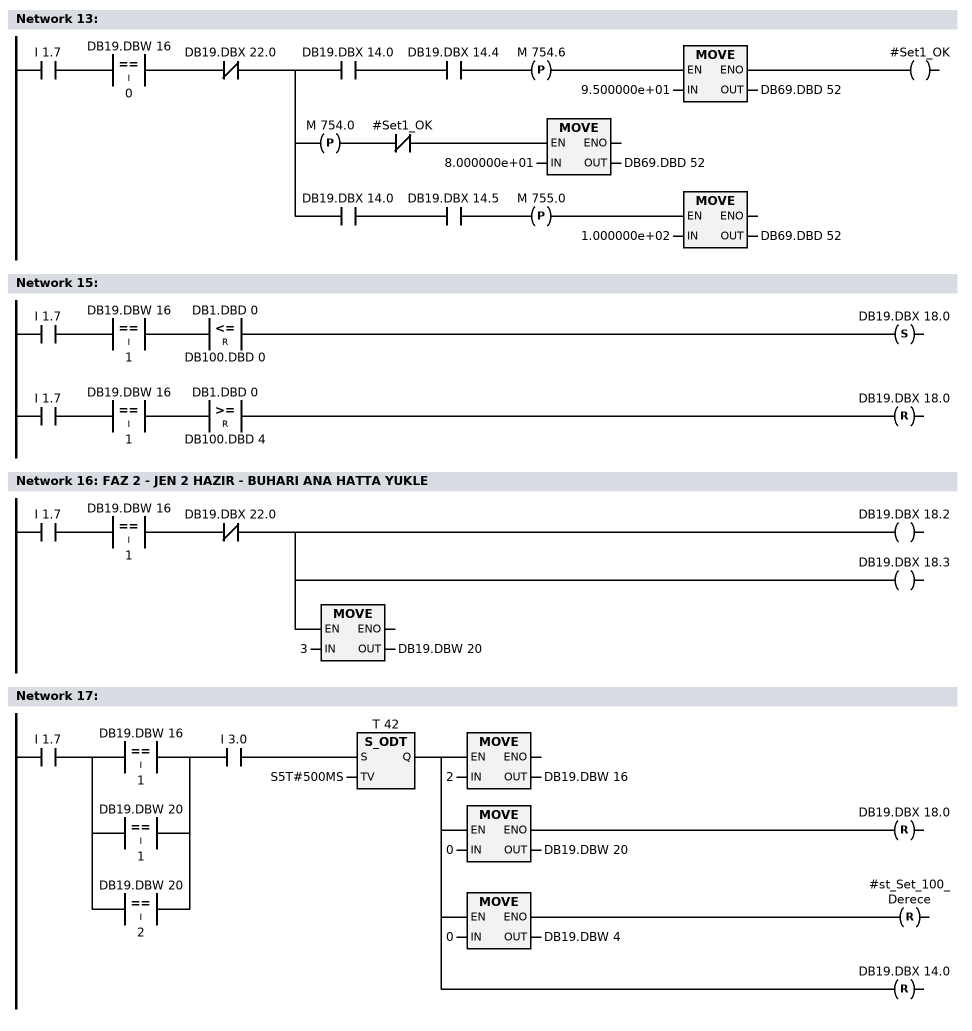
NETWORK
TITLE =
//-Sicaklik set 1 e geldiginde vana kapanma orani 5'e kadar düsüyor
//-Sicaklik set 2 e geldiginde vana kapanma orani 0'a kadar dusecek
//
//m754.0
//
      A     I 1.7;
      A(;
      L     DB19.DBW 16;
      L     0;
      ==I;
      );
      AN    DB19.DBX 22.0;
      =     L 2.0;
      A     L 2.0;
      A     DB19.DBX 14.0;
      A     DB19.DBX 14.4;
      FP    M 754.6;
      JNB   _00b;
      L     9.500000e+01;
      T     DB69.DBD 52;
      SET;
      SAVE;
      CLR;
_00b: A     BR;
      =     #Set1_OK;
      A     L 2.0;
      FP    M 754.0;
      AN    #Set1_OK;
      JNB   _00c;
      L     8.000000e+01;
      T     DB69.DBD 52;
_00c: NOP   0;
      A     L 2.0;
      A     DB19.DBX 14.0;
      A     DB19.DBX 14.5;
      FP    M 755.0;
      JNB   _00d;
      L     1.000000e+02;
      T     DB69.DBD 52;
_00d: NOP   0;
NETWORK
TITLE =
NETWORK
TITLE =
//FAZ - 2 MODUNA GEÇ
//1-BURLOR VE POMPA 4.5-5.5 BAR ARASINDA ÇALISIP DURACAK
      A     I 1.7;
      A(;
      L     DB19.DBW 16;
      L     1;
      ==I;
      );
      A(;
      L     DB1.DBD 0;
      L     DB100.DBD 0;
      <=R;
      );
      S     DB19.DBX 18.0;
      A     I 1.7;
      A(;
      L     DB19.DBW 16;
      L     1;
      ==I;
      );
      A(;
      L     DB1.DBD 0;
      L     DB100.DBD 4;
      >=R;
      );
      R     DB19.DBX 18.0;
      NOP   0;
NETWORK
TITLE = FAZ 2 - JEN 2 HAZIR - BUHARI ANA HATTA YUKLE
      A     I 1.7;
      A(;
      L     DB19.DBW 16;
      L     1;
      ==I;
      );
      AN    DB19.DBX 22.0;
      =     L 2.0;
      A     L 2.0;
      BLD   102;
      =     DB19.DBX 18.2;
      A     L 2.0;
      BLD   102;
      =     DB19.DBX 18.3;
      A     L 2.0;
      JNB   _00e;
      L     3;
      T     DB19.DBW 20;
_00e: NOP   0;
NETWORK
TITLE =
//FAZ 3 - GUVENLIK ONLEMLERI 
//1- 6 bar asildiginda -ok
//2- Baca 180 dereceyi gecerse -ok
//3- Su miktari min altina duserse -not ok
      A     I 1.7;
      A(;
      O(;
      L     DB19.DBW 16;
      L     1;
      ==I;
      );
      O(;
      L     DB19.DBW 20;
      L     1;
      ==I;
      );
      O(;
      L     DB19.DBW 20;
      L     2;
      ==I;
      );
      );
      A     I 3.0;
      L     S5T#500MS;
      SD    T 42;
      NOP   0;
      NOP   0;
      NOP   0;
      A     T 42;
      =     L 2.0;
      A     L 2.0;
      JNB   _00f;
      L     2;
      T     DB19.DBW 16;
_00f: NOP   0;
      A     L 2.0;
      JNB   _010;
      L     0;
      T     DB19.DBW 20;
      SET;
      SAVE;
      CLR;
_010: A     BR;
      R     DB19.DBX 18.0;
      A     L 2.0;
      JNB   _011;
      L     0;
      T     DB19.DBW 4;
      SET;
      SAVE;
      CLR;
_011: A     BR;
      R     #st_Set_100_Derece;
      A     L 2.0;
      BLD   102;
      R     DB19.DBX 14.0;
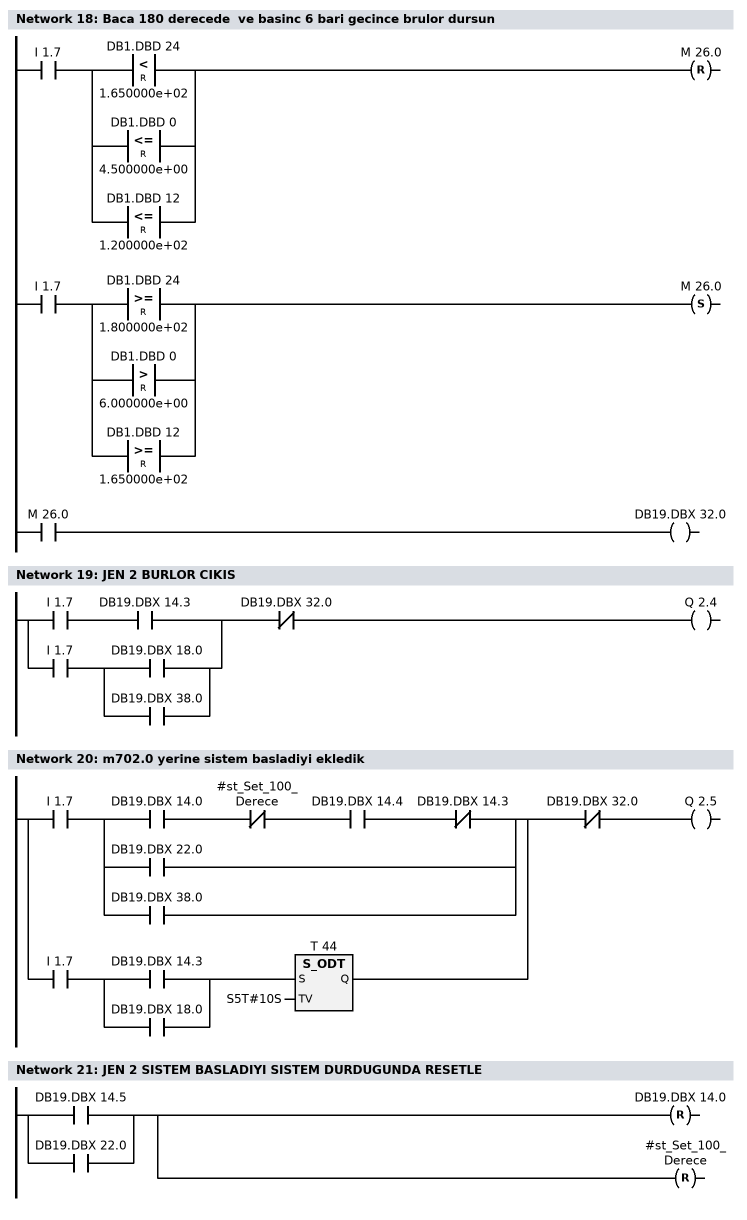
NETWORK
TITLE = Baca 180 derecede  ve basinc 6 bari gecince brulor dursun
      A     I 1.7;
      A(;
      O(;
      L     DB1.DBD 24;
      L     1.650000e+02;
      <R;
      );
      O(;
      L     DB1.DBD 0;
      L     4.500000e+00;
      <=R;
      );
      O(;
      L     DB1.DBD 12;
      L     1.200000e+02;
      <=R;
      );
      );
      R     M 26.0;
      A     I 1.7;
      A(;
      O(;
      L     DB1.DBD 24;
      L     1.800000e+02;
      >=R;
      );
      O(;
      L     DB1.DBD 0;
      L     6.000000e+00;
      >R;
      );
      O(;
      L     DB1.DBD 12;
      L     1.650000e+02;
      >=R;
      );
      );
      S     M 26.0;
      A     M 26.0;
      =     DB19.DBX 32.0;
NETWORK
TITLE = JEN 2 BURLOR CIKIS
      A(;
      A     I 1.7;
      A     DB19.DBX 14.3;
      O;
      A     I 1.7;
      A(;
      O     DB19.DBX 18.0;
      O     DB19.DBX 38.0;
      );
      );
      AN    DB19.DBX 32.0;
      =     Q 2.4;
NETWORK
TITLE = m702.0 yerine sistem basladiyi ekledik
//q2.5 motor çikisi
      A(;
      A     I 1.7;
      A(;
      A     DB19.DBX 14.0;
      AN    #st_Set_100_Derece;
      A     DB19.DBX 14.4;
      AN    DB19.DBX 14.3;
      O     DB19.DBX 22.0;
      O     DB19.DBX 38.0;
      );
      O(;
      A     I 1.7;
      A(;
      O     DB19.DBX 14.3;
      O     DB19.DBX 18.0;
      );
      L     S5T#10S;
      SD    T 44;
      NOP   0;
      NOP   0;
      NOP   0;
      A     T 44;
      );
      );
      AN    DB19.DBX 32.0;
      =     Q 2.5;
NETWORK
TITLE = JEN 2 SISTEM BASLADIYI SISTEM DURDUGUNDA RESETLE
      O     DB19.DBX 14.5;
      O     DB19.DBX 22.0;
      R     DB19.DBX 14.0;
      R     #st_Set_100_Derece;
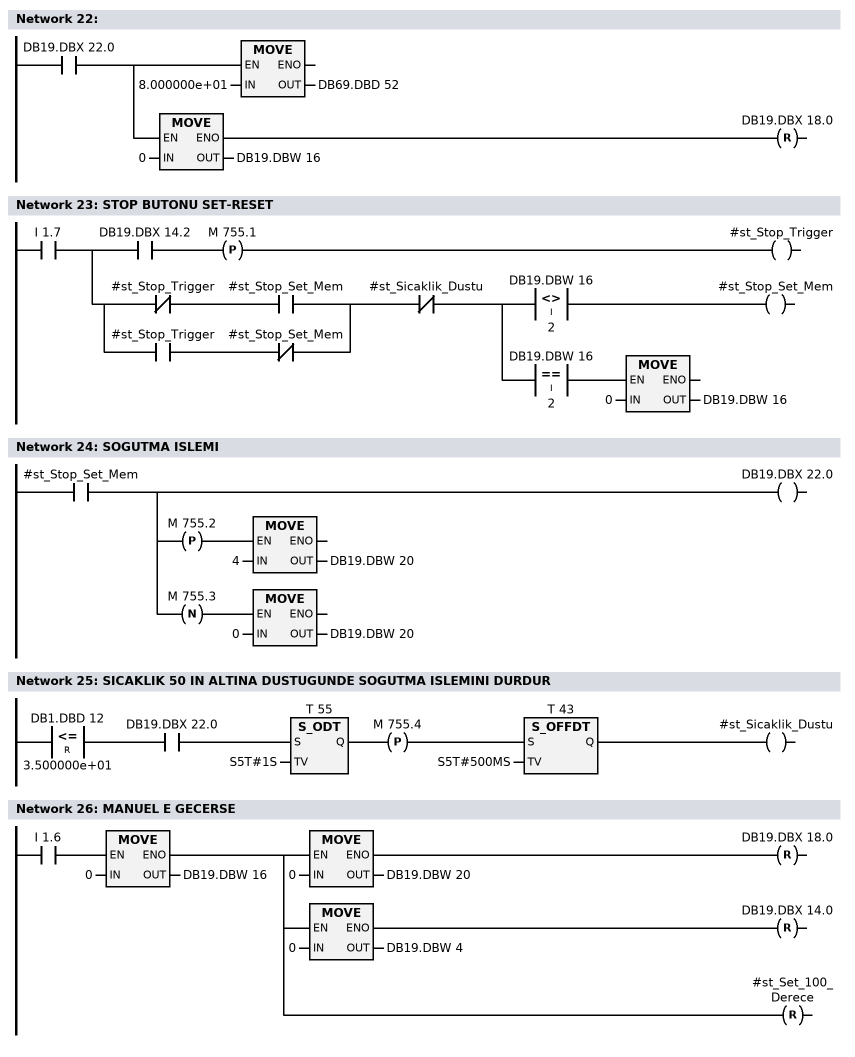
NETWORK
TITLE =
      A     DB19.DBX 22.0;
      =     L 2.0;
      A     L 2.0;
      JNB   _012;
      L     8.000000e+01;
      T     DB69.DBD 52;
_012: NOP   0;
      A     L 2.0;
      JNB   _013;
      L     0;
      T     DB19.DBW 16;
      SET;
      SAVE;
      CLR;
_013: A     BR;
      R     DB19.DBX 18.0;
NETWORK
TITLE = STOP BUTONU SET-RESET
      A     I 1.7;
      =     L 2.0;
      A     L 2.0;
      A     DB19.DBX 14.2;
      FP    M 755.1;
      =     #st_Stop_Trigger;
      A     L 2.0;
      A(;
      AN    #st_Stop_Trigger;
      A     #st_Stop_Set_Mem;
      O;
      A     #st_Stop_Trigger;
      AN    #st_Stop_Set_Mem;
      );
      AN    #st_Sicaklik_Dustu;
      =     L 2.1;
      A     L 2.1;
      A(;
      L     DB19.DBW 16;
      L     2;
      <>I;
      );
      =     #st_Stop_Set_Mem;
      A     L 2.1;
      A(;
      L     DB19.DBW 16;
      L     2;
      ==I;
      );
      JNB   _014;
      L     0;
      T     DB19.DBW 16;
_014: NOP   0;
NETWORK
TITLE = SOGUTMA ISLEMI
      A     #st_Stop_Set_Mem;
      =     L 2.0;
      A     L 2.0;
      BLD   102;
      =     DB19.DBX 22.0;
      A     L 2.0;
      FP    M 755.2;
      JNB   _015;
      L     4;
      T     DB19.DBW 20;
_015: NOP   0;
      A     L 2.0;
      FN    M 755.3;
      JNB   _016;
      L     0;
      T     DB19.DBW 20;
_016: NOP   0;
NETWORK
TITLE = SICAKLIK 50 IN ALTINA DUSTUGUNDE SOGUTMA ISLEMINI DURDUR
      A(;
      A(;
      L     DB1.DBD 12;
      L     3.500000e+01;
      <=R;
      );
      A     DB19.DBX 22.0;
      L     S5T#1S;
      SD    T 55;
      NOP   0;
      NOP   0;
      NOP   0;
      A     T 55;
      );
      FP    M 755.4;
      L     S5T#500MS;
      SF    T 43;
      NOP   0;
      NOP   0;
      NOP   0;
      A     T 43;
      =     #st_Sicaklik_Dustu;
NETWORK
TITLE = MANUEL E GECERSE
      A     I 1.6;
      JNB   _017;
      L     0;
      T     DB19.DBW 16;
      SET;
      SAVE;
      CLR;
_017: A     BR;
      =     L 2.0;
      A     L 2.0;
      JNB   _018;
      L     0;
      T     DB19.DBW 20;
      SET;
      SAVE;
      CLR;
_018: A     BR;
      R     DB19.DBX 18.0;
      A     L 2.0;
      JNB   _019;
      L     0;
      T     DB19.DBW 4;
      SET;
      SAVE;
      CLR;
_019: A     BR;
      R     DB19.DBX 14.0;
      A     L 2.0;
      BLD   102;
      R     #st_Set_100_Derece;
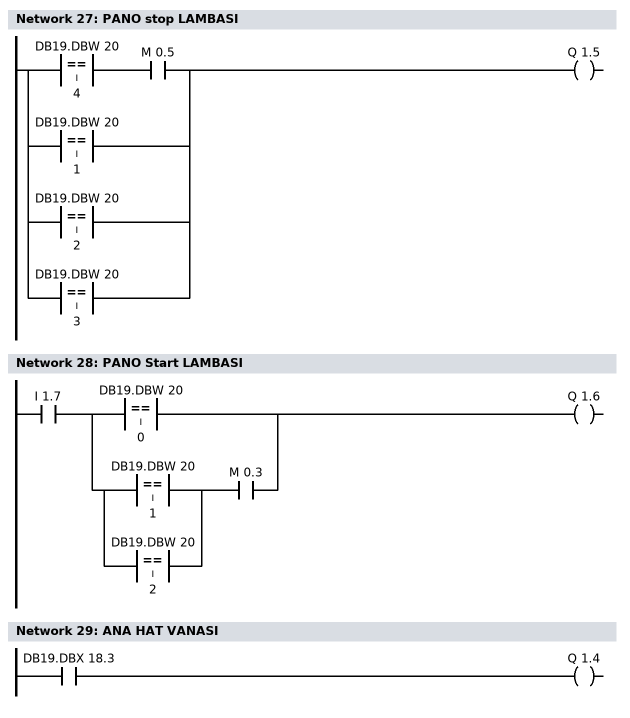
NETWORK
TITLE = PANO stop LAMBASI
      A(;
      L     DB19.DBW 20;
      L     4;
      ==I;
      );
      A     M 0.5;
      O(;
      L     DB19.DBW 20;
      L     1;
      ==I;
      );
      O(;
      L     DB19.DBW 20;
      L     2;
      ==I;
      );
      O(;
      L     DB19.DBW 20;
      L     3;
      ==I;
      );
      =     Q 1.5;
NETWORK
TITLE = PANO Start LAMBASI
      A     I 1.7;
      A(;
      O(;
      L     DB19.DBW 20;
      L     0;
      ==I;
      );
      O;
      A(;
      O(;
      L     DB19.DBW 20;
      L     1;
      ==I;
      );
      O(;
      L     DB19.DBW 20;
      L     2;
      ==I;
      );
      );
      A     M 0.3;
      );
      =     Q 1.6;
NETWORK
TITLE = ANA HAT VANASI 
      A     DB19.DBX 18.3;
      =     Q 1.4;
END_FUNCTION_BLOCK

FUNCTION_BLOCK FB 99
//PIW 286 - Jen 2 Basinc
//PIW 288 - Jen 2 Buhar Sicakligi
//PQW 278 - Jen 2 Baca Sicakligi
VERSION : 0.1
VAR
  Rising_Status : BOOL ;
  Rising_Startup : BOOL ;
  Set_100_Derece : BOOL ;
  Rising_After_Stop : BOOL ;
  Set1_OK : BOOL ;
  Rising_Status_3 : BOOL ;
  Rising_Status_4 : BOOL ;
  Rising_100_dere_reset : BOOL ;
  Ris_Set1_ok_95 : BOOL ;
  Ris_Set2_ok_100 : BOOL ;
END_VAR
BEGIN
NETWORK
TITLE = Analog Çeviriler
      A     M 100.0;
      =     L 0.0;
      BLD   103;
      A(;
      A     M 100.0;
      =     L 0.1;
      BLD   103;
      CALL  FC 105 (
           $1                       := P#P 286.0,
           $2                       := L#1092616192,
           $3                       := L#0,
           $4                       := L 0.1,
           $5                       := DB1.DBW 10,
           $6                       := DB1.DBD 4);
      A     BR;
      );
      JNB   _001;
      CALL  FC 105 (
           $1                       := P#P 288.0,
           $2                       := L#1128792064,
           $3                       := L#0,
           $4                       := L 0.0,
           $5                       := DB1.DBW 22,
           $6                       := DB1.DBD 16);
_001: NOP   0;
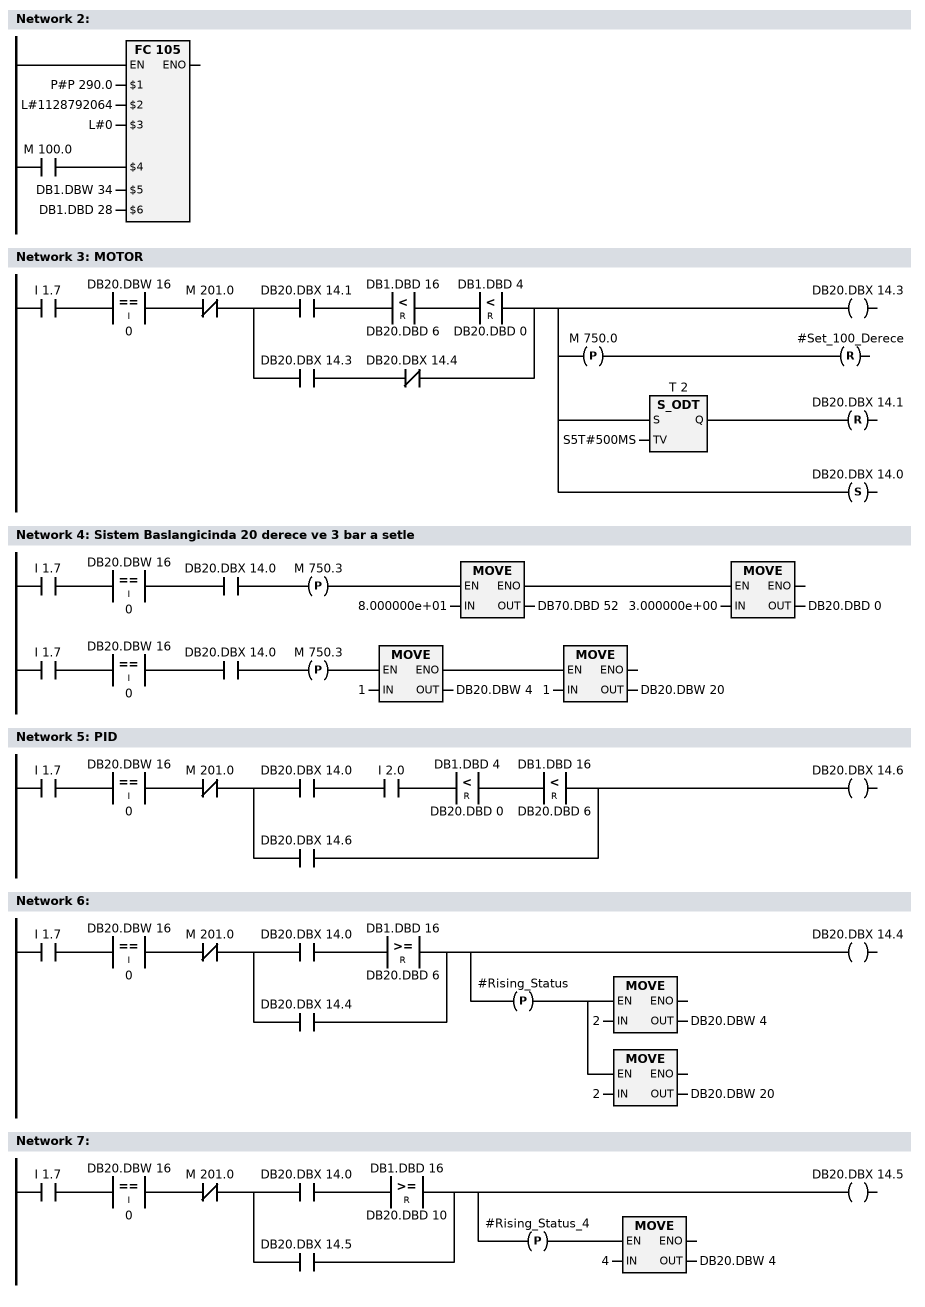
NETWORK
TITLE =
      A     M 100.0;
      =     L 0.0;
      BLD   103;
      CALL  FC 105 (
           $1                       := P#P 290.0,
           $2                       := L#1128792064,
           $3                       := L#0,
           $4                       := L 0.0,
           $5                       := DB1.DBW 34,
           $6                       := DB1.DBD 28);
      NOP   0;
NETWORK
TITLE = MOTOR
      A     I 1.7;
      A(;
      L     DB20.DBW 16;
      L     0;
      ==I;
      );
      AN    M 201.0;
      A(;
      A     DB20.DBX 14.1;
      A(;
      L     DB1.DBD 16;
      L     DB20.DBD 6;
      <R;
      );
      A(;
      L     DB1.DBD 4;
      L     DB20.DBD 0;
      <R;
      );
      O;
      A     DB20.DBX 14.3;
      AN    DB20.DBX 14.4;
      );
      =     L 0.0;
      A     L 0.0;
      BLD   102;
      =     DB20.DBX 14.3;
      A     L 0.0;
      FP    M 750.0;
      R     #Set_100_Derece;
      A     L 0.0;
      L     S5T#500MS;
      SD    T 2;
      NOP   0;
      NOP   0;
      NOP   0;
      A     T 2;
      R     DB20.DBX 14.1;
      A     L 0.0;
      BLD   102;
      S     DB20.DBX 14.0;
NETWORK
TITLE = Sistem Baslangicinda 20 derece ve 3 bar a setle
      A     I 1.7;
      A(;
      L     DB20.DBW 16;
      L     0;
      ==I;
      );
      A     DB20.DBX 14.0;
      FP    M 750.3;
      =     L 0.0;
      A(;
      A     L 0.0;
      JNB   _002;
      L     8.000000e+01;
      T     DB70.DBD 52;
      SET;
      SAVE;
      CLR;
_002: A     BR;
      );
      JNB   _003;
      L     3.000000e+00;
      T     DB20.DBD 0;
_003: NOP   0;
      A(;
      A     L 0.0;
      JNB   _004;
      L     1;
      T     DB20.DBW 4;
      SET;
      SAVE;
      CLR;
_004: A     BR;
      );
      JNB   _005;
      L     1;
      T     DB20.DBW 20;
_005: NOP   0;
NETWORK
TITLE = PID
      A     I 1.7;
      A(;
      L     DB20.DBW 16;
      L     0;
      ==I;
      );
      AN    M 201.0;
      A(;
      A     DB20.DBX 14.0;
      A     I 2.0;
      A(;
      L     DB1.DBD 4;
      L     DB20.DBD 0;
      <R;
      );
      A(;
      L     DB1.DBD 16;
      L     DB20.DBD 6;
      <R;
      );
      O     DB20.DBX 14.6;
      );
      =     DB20.DBX 14.6;
NETWORK
TITLE =
      A     I 1.7;
      A(;
      L     DB20.DBW 16;
      L     0;
      ==I;
      );
      AN    M 201.0;
      A(;
      A     DB20.DBX 14.0;
      A(;
      L     DB1.DBD 16;
      L     DB20.DBD 6;
      >=R;
      );
      O     DB20.DBX 14.4;
      );
      =     L 0.0;
      A     L 0.0;
      BLD   102;
      =     DB20.DBX 14.4;
      A     L 0.0;
      FP    #Rising_Status;
      =     L 0.1;
      A     L 0.1;
      JNB   _006;
      L     2;
      T     DB20.DBW 4;
_006: NOP   0;
      A     L 0.1;
      JNB   _007;
      L     2;
      T     DB20.DBW 20;
_007: NOP   0;
NETWORK
TITLE =
      A     I 1.7;
      A(;
      L     DB20.DBW 16;
      L     0;
      ==I;
      );
      AN    M 201.0;
      A(;
      A     DB20.DBX 14.0;
      A(;
      L     DB1.DBD 16;
      L     DB20.DBD 10;
      >=R;
      );
      O     DB20.DBX 14.5;
      );
      =     L 0.0;
      A     L 0.0;
      BLD   102;
      =     DB20.DBX 14.5;
      A     L 0.0;
      FP    #Rising_Status_4;
      JNB   _008;
      L     4;
      T     DB20.DBW 4;
_008: NOP   0;
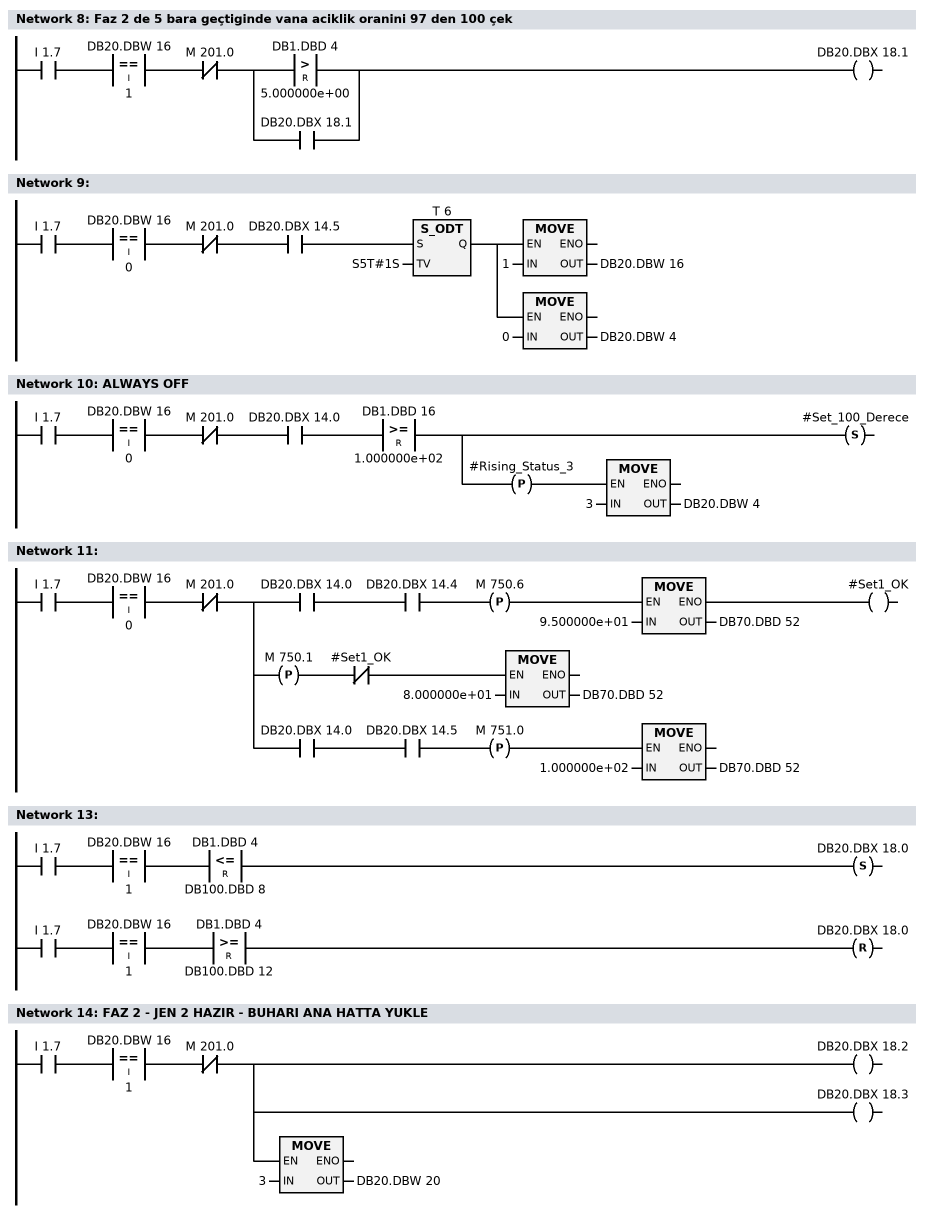
NETWORK
TITLE = Faz 2 de 5 bara geçtiginde vana aciklik oranini 97 den 100 çek
      A     I 1.7;
      A(;
      L     DB20.DBW 16;
      L     1;
      ==I;
      );
      AN    M 201.0;
      A(;
      O(;
      L     DB1.DBD 4;
      L     5.000000e+00;
      >R;
      );
      O     DB20.DBX 18.1;
      );
      =     DB20.DBX 18.1;
NETWORK
TITLE =
//SET 2 SICAKLIGINDAN SONRA FAZ 2 E GEC
      A     I 1.7;
      A(;
      L     DB20.DBW 16;
      L     0;
      ==I;
      );
      AN    M 201.0;
      A     DB20.DBX 14.5;
      L     S5T#1S;
      SD    T 6;
      NOP   0;
      NOP   0;
      NOP   0;
      A     T 6;
      =     L 0.0;
      A     L 0.0;
      JNB   _009;
      L     1;
      T     DB20.DBW 16;
_009: NOP   0;
      A     L 0.0;
      JNB   _00a;
      L     0;
      T     DB20.DBW 4;
_00a: NOP   0;
NETWORK
TITLE = ALWAYS OFF
//Pompa 100 derecede duracak
      A     I 1.7;
      A(;
      L     DB20.DBW 16;
      L     0;
      ==I;
      );
      AN    M 201.0;
      A     DB20.DBX 14.0;
      A(;
      L     DB1.DBD 16;
      L     1.000000e+02;
      >=R;
      );
      =     L 0.0;
      A     L 0.0;
      BLD   102;
      S     #Set_100_Derece;
      A     L 0.0;
      FP    #Rising_Status_3;
      JNB   _00b;
      L     3;
      T     DB20.DBW 4;
_00b: NOP   0;
NETWORK
TITLE =
//-Sicaklik set 1 e geldiginde vana kapanma orani 5'e kadar düsüyor
//-Sicaklik set 2 e geldiginde vana kapanma orani 0'a kadar dusecek
      A     I 1.7;
      A(;
      L     DB20.DBW 16;
      L     0;
      ==I;
      );
      AN    M 201.0;
      =     L 0.0;
      A     L 0.0;
      A     DB20.DBX 14.0;
      A     DB20.DBX 14.4;
      FP    M 750.6;
      JNB   _00c;
      L     9.500000e+01;
      T     DB70.DBD 52;
      SET;
      SAVE;
      CLR;
_00c: A     BR;
      =     #Set1_OK;
      A     L 0.0;
      FP    M 750.1;
      AN    #Set1_OK;
      JNB   _00d;
      L     8.000000e+01;
      T     DB70.DBD 52;
_00d: NOP   0;
      A     L 0.0;
      A     DB20.DBX 14.0;
      A     DB20.DBX 14.5;
      FP    M 751.0;
      JNB   _00e;
      L     1.000000e+02;
      T     DB70.DBD 52;
_00e: NOP   0;
NETWORK
TITLE =
NETWORK
TITLE =
//FAZ - 2 MODUNA GEÇ
//1-BURLOR VE POMPA 4.5-5.5 BAR ARASINDA ÇALISIP DURACAK
      A     I 1.7;
      A(;
      L     DB20.DBW 16;
      L     1;
      ==I;
      );
      A(;
      L     DB1.DBD 4;
      L     DB100.DBD 8;
      <=R;
      );
      S     DB20.DBX 18.0;
      A     I 1.7;
      A(;
      L     DB20.DBW 16;
      L     1;
      ==I;
      );
      A(;
      L     DB1.DBD 4;
      L     DB100.DBD 12;
      >=R;
      );
      R     DB20.DBX 18.0;
      NOP   0;
NETWORK
TITLE = FAZ 2 - JEN 2 HAZIR - BUHARI ANA HATTA YUKLE
      A     I 1.7;
      A(;
      L     DB20.DBW 16;
      L     1;
      ==I;
      );
      AN    M 201.0;
      =     L 0.0;
      A     L 0.0;
      BLD   102;
      =     DB20.DBX 18.2;
      A     L 0.0;
      BLD   102;
      =     DB20.DBX 18.3;
      A     L 0.0;
      JNB   _00f;
      L     3;
      T     DB20.DBW 20;
_00f: NOP   0;
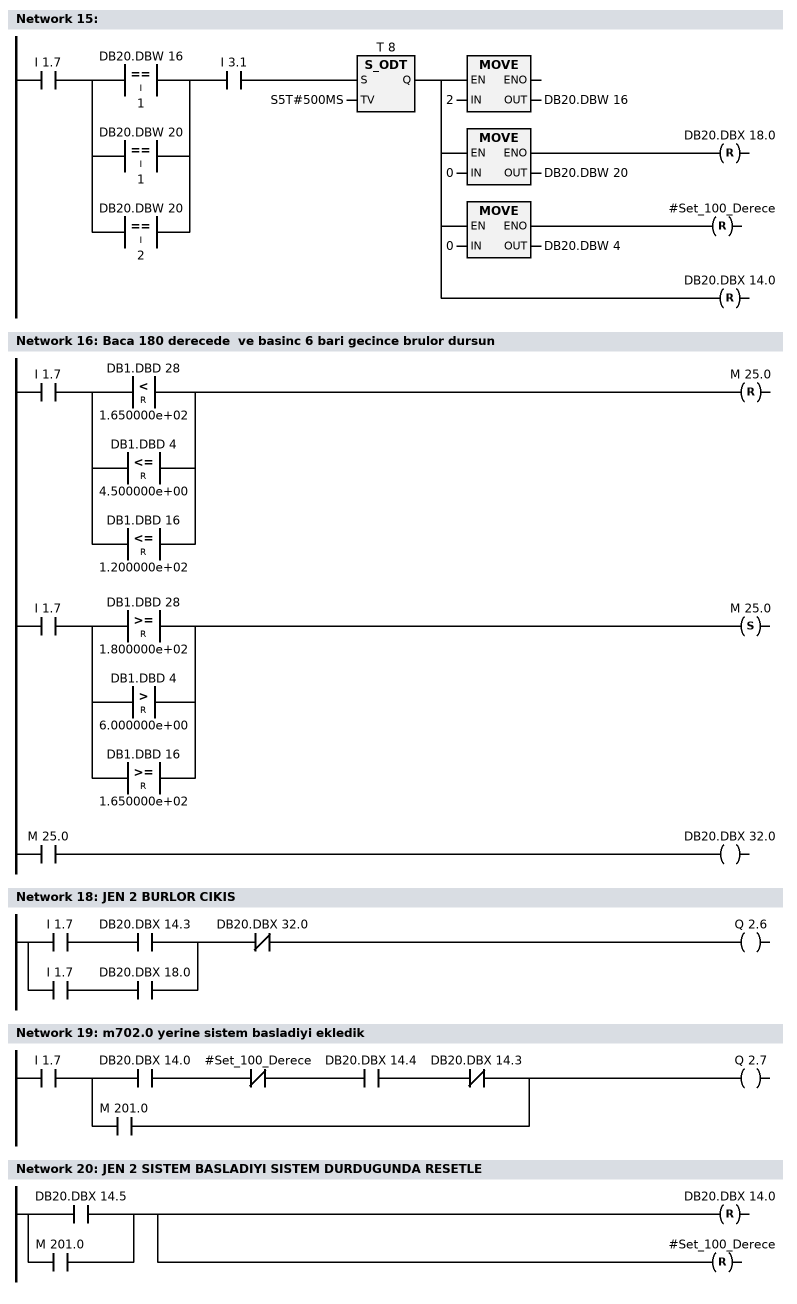
NETWORK
TITLE =
//FAZ 3 - GUVENLIK ONLEMLERI 
//1- 6 bar asildiginda -ok
//2- Baca 180 dereceyi gecerse -ok
//3- Su miktari min altina duserse -ok
      A     I 1.7;
      A(;
      O(;
      L     DB20.DBW 16;
      L     1;
      ==I;
      );
      O(;
      L     DB20.DBW 20;
      L     1;
      ==I;
      );
      O(;
      L     DB20.DBW 20;
      L     2;
      ==I;
      );
      );
      A     I 3.1;
      L     S5T#500MS;
      SD    T 8;
      NOP   0;
      NOP   0;
      NOP   0;
      A     T 8;
      =     L 0.0;
      A     L 0.0;
      JNB   _010;
      L     2;
      T     DB20.DBW 16;
_010: NOP   0;
      A     L 0.0;
      JNB   _011;
      L     0;
      T     DB20.DBW 20;
      SET;
      SAVE;
      CLR;
_011: A     BR;
      R     DB20.DBX 18.0;
      A     L 0.0;
      JNB   _012;
      L     0;
      T     DB20.DBW 4;
      SET;
      SAVE;
      CLR;
_012: A     BR;
      R     #Set_100_Derece;
      A     L 0.0;
      BLD   102;
      R     DB20.DBX 14.0;
NETWORK
TITLE = Baca 180 derecede  ve basinc 6 bari gecince brulor dursun
      A     I 1.7;
      A(;
      O(;
      L     DB1.DBD 28;
      L     1.650000e+02;
      <R;
      );
      O(;
      L     DB1.DBD 4;
      L     4.500000e+00;
      <=R;
      );
      O(;
      L     DB1.DBD 16;
      L     1.200000e+02;
      <=R;
      );
      );
      R     M 25.0;
      A     I 1.7;
      A(;
      O(;
      L     DB1.DBD 28;
      L     1.800000e+02;
      >=R;
      );
      O(;
      L     DB1.DBD 4;
      L     6.000000e+00;
      >R;
      );
      O(;
      L     DB1.DBD 16;
      L     1.650000e+02;
      >=R;
      );
      );
      S     M 25.0;
      A     M 25.0;
      =     DB20.DBX 32.0;
NETWORK
TITLE =
NETWORK
TITLE = JEN 2 BURLOR CIKIS
      A(;
      A     I 1.7;
      A     DB20.DBX 14.3;
      O;
      A     I 1.7;
      A     DB20.DBX 18.0;
      );
      AN    DB20.DBX 32.0;
      =     Q 2.6;
NETWORK
TITLE = m702.0 yerine sistem basladiyi ekledik
      A     I 1.7;
      A(;
      A     DB20.DBX 14.0;
      AN    #Set_100_Derece;
      A     DB20.DBX 14.4;
      AN    DB20.DBX 14.3;
      O     M 201.0;
      );
      =     Q 2.7;
NETWORK
TITLE = JEN 2 SISTEM BASLADIYI SISTEM DURDUGUNDA RESETLE
      O     DB20.DBX 14.5;
      O     M 201.0;
      R     DB20.DBX 14.0;
      R     #Set_100_Derece;
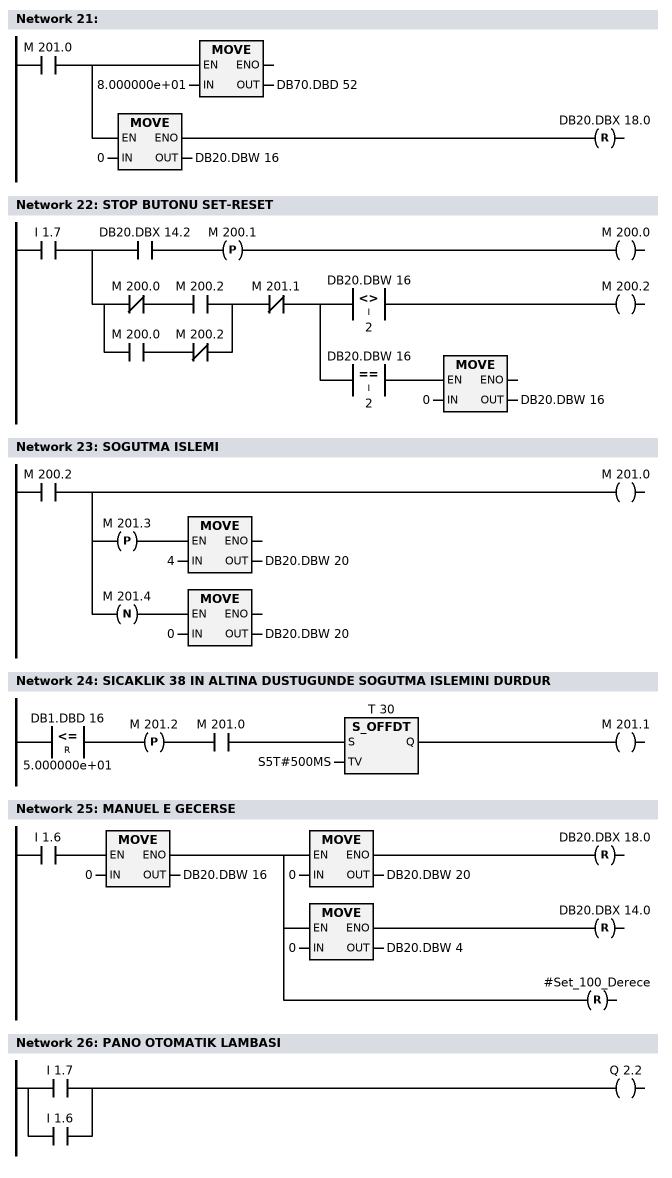
NETWORK
TITLE =
      A     M 201.0;
      =     L 0.0;
      A     L 0.0;
      JNB   _013;
      L     8.000000e+01;
      T     DB70.DBD 52;
_013: NOP   0;
      A     L 0.0;
      JNB   _014;
      L     0;
      T     DB20.DBW 16;
      SET;
      SAVE;
      CLR;
_014: A     BR;
      R     DB20.DBX 18.0;
NETWORK
TITLE = STOP BUTONU SET-RESET
      A     I 1.7;
      =     L 0.0;
      A     L 0.0;
      A     DB20.DBX 14.2;
      FP    M 200.1;
      =     M 200.0;
      A     L 0.0;
      A(;
      AN    M 200.0;
      A     M 200.2;
      O;
      A     M 200.0;
      AN    M 200.2;
      );
      AN    M 201.1;
      =     L 0.1;
      A     L 0.1;
      A(;
      L     DB20.DBW 16;
      L     2;
      <>I;
      );
      =     M 200.2;
      A     L 0.1;
      A(;
      L     DB20.DBW 16;
      L     2;
      ==I;
      );
      JNB   _015;
      L     0;
      T     DB20.DBW 16;
_015: NOP   0;
NETWORK
TITLE = SOGUTMA ISLEMI
      A     M 200.2;
      =     L 0.0;
      A     L 0.0;
      BLD   102;
      =     M 201.0;
      A     L 0.0;
      FP    M 201.3;
      JNB   _016;
      L     4;
      T     DB20.DBW 20;
_016: NOP   0;
      A     L 0.0;
      FN    M 201.4;
      JNB   _017;
      L     0;
      T     DB20.DBW 20;
_017: NOP   0;
NETWORK
TITLE = SICAKLIK 38 IN ALTINA DUSTUGUNDE SOGUTMA ISLEMINI DURDUR
      A(;
      L     DB1.DBD 16;
      L     5.000000e+01;
      <=R;
      );
      FP    M 201.2;
      A     M 201.0;
      L     S5T#500MS;
      SF    T 30;
      NOP   0;
      NOP   0;
      NOP   0;
      A     T 30;
      =     M 201.1;
NETWORK
TITLE = MANUEL E GECERSE
      A     I 1.6;
      JNB   _018;
      L     0;
      T     DB20.DBW 16;
      SET;
      SAVE;
      CLR;
_018: A     BR;
      =     L 0.0;
      A     L 0.0;
      JNB   _019;
      L     0;
      T     DB20.DBW 20;
      SET;
      SAVE;
      CLR;
_019: A     BR;
      R     DB20.DBX 18.0;
      A     L 0.0;
      JNB   _01a;
      L     0;
      T     DB20.DBW 4;
      SET;
      SAVE;
      CLR;
_01a: A     BR;
      R     DB20.DBX 14.0;
      A     L 0.0;
      BLD   102;
      R     #Set_100_Derece;
NETWORK
TITLE = PANO OTOMATIK LAMBASI
      O     I 1.7;
      O     I 1.6;
      =     Q 2.2;
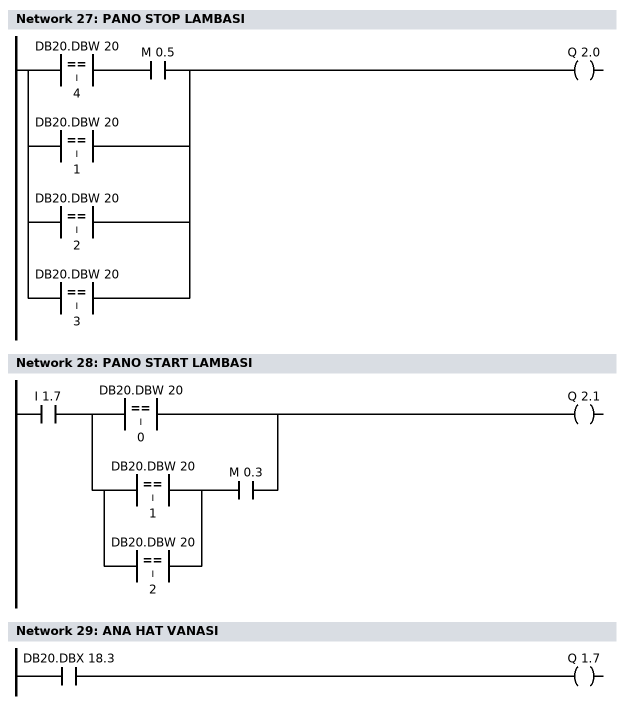
NETWORK
TITLE = PANO STOP LAMBASI
//1- Buhar hazýrlaniyor
//2- set 1 e ulasti
//3- Basinci Stabil tutma
//4- Sogutma
      A(;
      L     DB20.DBW 20;
      L     4;
      ==I;
      );
      A     M 0.5;
      O(;
      L     DB20.DBW 20;
      L     1;
      ==I;
      );
      O(;
      L     DB20.DBW 20;
      L     2;
      ==I;
      );
      O(;
      L     DB20.DBW 20;
      L     3;
      ==I;
      );
      =     Q 2.0;
NETWORK
TITLE = PANO START LAMBASI
      A     I 1.7;
      A(;
      O(;
      L     DB20.DBW 20;
      L     0;
      ==I;
      );
      O;
      A(;
      O(;
      L     DB20.DBW 20;
      L     1;
      ==I;
      );
      O(;
      L     DB20.DBW 20;
      L     2;
      ==I;
      );
      );
      A     M 0.3;
      );
      =     Q 2.1;
NETWORK
TITLE = ANA HAT VANASI 
      A     DB20.DBX 18.3;
      =     Q 1.7;
END_FUNCTION_BLOCK

FUNCTION FC 1 : VOID
VERSION : 0.0
VAR_INPUT
  iTimeET : TIME ;
  iIstenileSure : S5TIME ;
END_VAR
VAR_OUTPUT
  oOUT : DINT ;
END_VAR
VAR_TEMP
  vTemp : DINT ;
  vValue : DINT ;
  vValue2 : DINT ;
  vIstenilenTime : TIME ;
  vIstenilenDint : DINT ;
END_VAR
BEGIN
// body was compiled from an SCL source; compiled code not shown
END_FUNCTION

// FC 33: know-how protected block, not included

// FC 105: know-how protected block, not included

// FC 106: know-how protected block, not included

DATA_BLOCK DB 1
VERSION : 0.1
  STRUCT
   JEN1_BASINC_ANLIK : REAL ;
   JEN2_BASINC_ANLIK : REAL ;
   JEN1_BASINC_RET_VAL : WORD ;
   JEN2_BASINC_RET_VAL : WORD ;
   JEN1_IC_SICAKLIK_ANLIK : REAL ;
   JEN2_IC_SICAKLIK_ANLIK : REAL ;
   JEN1_IC_SICAKLIK_RET_VAL : WORD ;
   JEN2_IC_SICAKLIK_RET_VAL : WORD ;
   JEN1_BACA_SICAKLIK_ANLIK : REAL ;
   JEN2_BACA_SICAKLIK_ANLIK : REAL ;
   JEN1_BACA_SICAKLIK_RET_V : WORD ;
   JEN2_BACA_SICAKLIK_RET_V : WORD ;
   HAT_BASINCI_RET_V : WORD ;
   HAT_BASINCI_ANLIK : REAL ;
   HAVA_BASINCI_RET_V : WORD ;
   HAVA_BASINCI_ANLIK : REAL ;
   HAT_BASINCI_YETERLI : BOOL ;
  END_STRUCT ;	
BEGIN
END_DATA_BLOCK

DATA_BLOCK DB 2
VERSION : 0.1
  STRUCT
   JEN_EMNIYET_BASINCI : REAL ;
   JEN_EMNIYET_SICAKLIGI : REAL ;
   OTO_EMNIYET_BASINCI : REAL ;
   OTO_EMNIYET_SICAKLIGI : REAL ;
   OTO_ISLEM_BITTI_VANA_AC : BOOL ;
   OTO_JEN_DURDU : REAL ;
  END_STRUCT ;	
BEGIN
END_DATA_BLOCK

DATA_BLOCK DB 5
AUTHOR : SIMATIC
FAMILY : IEC_TC
VERSION : 0.0
SFB 4
BEGIN
END_DATA_BLOCK

DATA_BLOCK DB 6
AUTHOR : SIMATIC
FAMILY : IEC_TC
VERSION : 0.0
SFB 4
BEGIN
END_DATA_BLOCK

DATA_BLOCK DB 7
AUTHOR : SIMATIC
FAMILY : IEC_TC
VERSION : 0.0
SFB 4
BEGIN
END_DATA_BLOCK

DATA_BLOCK DB 8
AUTHOR : SIMATIC
FAMILY : IEC_TC
VERSION : 0.0
SFB 4
BEGIN
END_DATA_BLOCK

DATA_BLOCK DB 9
AUTHOR : SIMATIC
FAMILY : IEC_TC
VERSION : 0.0
SFB 4
BEGIN
END_DATA_BLOCK

DATA_BLOCK DB 10
AUTHOR : SIMATIC
FAMILY : IEC_TC
VERSION : 0.0
SFB 4
BEGIN
END_DATA_BLOCK

DATA_BLOCK DB 14
VERSION : 0.0
FB 3
BEGIN
END_DATA_BLOCK

DATA_BLOCK DB 15
VERSION : 0.0
FB 2
BEGIN
END_DATA_BLOCK

DATA_BLOCK DB 17
VERSION : 0.1
  STRUCT
   IN_STATUS : INT ;
   IN_JEN_OK : BOOL ;
   IN_DIGER_KAZ_TRANS_HAZIR : BOOL ;
   IN_PISIM_SURESI : S5TIME ;
   IN_SCALE_BASINC_PER : INT ;
   IN_SET_BASINC : REAL ;
   IN_DIGER_KAZAN_BASINCI : REAL ;
   O_PID_MAN_ON : BOOL ;
   O_PID_MAN : REAL ;
   O_TRANSFER_YAPILIYOR : BOOL ;
   O_SCALE_BASINC_RET_VAL : WORD ;
   O_SCALE_BASINC_OUT : REAL ;
   O_TRANSFERE_HAZIR : BOOL ;
   O_SCALE_SICAKLIK_RET_VAL : WORD ;
   O_SCALE_SICAKLIK_OUT : REAL ;
   IN_SCALE_SICAKLIK_PER : INT ;
   O_KAZAN_BOSALTIMDA : BOOL ;
   IN_DIGER_KAZ_BOSALTIMDA : BOOL ;
   IN_DIGER_KAZ_TRANSFERDE : BOOL ;
   O_PISIM_BASLADI : BOOL ;
   PISIM_GECEN_SURE_TIME : TIME ;
   PISIM_GECEN_SURE_DINT : DINT ;
   PROSES_SURESI_TIME : TIME ;
   PROSES_SURESI_DINT : DINT ;
   BEKLEME_SURESI_TIME : TIME ;
   BEKLEME_SURESI_DINT : DINT ;
  END_STRUCT ;	
BEGIN
END_DATA_BLOCK

DATA_BLOCK DB 18
VERSION : 0.1
  STRUCT
   IN_STATUS : INT ;
   IN_JEN_OK : BOOL ;
   IN_DIGER_KAZ_TRANS_HAZIR : BOOL ;
   IN_PISIM_SURESI : S5TIME ;
   IN_SCALE_BASINC_PER : INT ;
   IN_SET_BASINC : REAL ;
   IN_DIGER_KAZAN_BASINCI : REAL ;
   O_PID_MAN_ON : BOOL ;
   O_PID_MAN : REAL ;
   O_TRANSFER_YAPILIYOR : BOOL ;
   O_SCALE_BASINC_RET_VAL : WORD ;
   O_SCALE_BASINC_OUT : REAL ;
   O_TRANSFERE_HAZIR : BOOL ;
   O_SCALE_SICAKLIK_RET_VAL : WORD ;
   O_SCALE_SICAKLIK_OUT : REAL ;
   IN_SCALE_SICAKLIK_PER : INT ;
   O_KAZAN_BOSALTIMDA : BOOL ;
   IN_DIGER_KAZ_BOSALTIMDA : BOOL ;
   IN_DIGER_KAZ_TRANSFERDE : BOOL ;
   O_PISIM_BASLADI : BOOL ;
   PISIM_GECEN_SURE_TIME : TIME ;
   PISIM_GECEN_SURE_DINT : DINT ;
   PROSES_SURESI_TIM : TIME ;
   PROSES_SURESI_DINT : DINT ;
   BEKLEME_SURESI_TIME : TIME ;
   BEKLEME_SURESI_DINT : DINT ;
  END_STRUCT ;	
BEGIN
END_DATA_BLOCK

DATA_BLOCK DB 19
VERSION : 0.1
  STRUCT
   BASINC_SET_POINT : REAL ;
   STATUS : INT ;
   SICAKLIK_SET_POINT_1 : REAL ;
   SICAKLIK_SET_POINT_2 : REAL ;
   SISTEM_BASLADI : BOOL ;
   EKRAN_START : BOOL ;
   EKRAN_STOP : BOOL ;
   OUT_BURLOR_MOT_START : BOOL ;
   SICAKLIK_SET1_OK : BOOL ;
   SICAKLIK_SET2_OK : BOOL ;
   OUT_PID_START : BOOL ;
   FAZ_GECISI_STATUS : INT ;
   FAZ_2_SET_RESET : BOOL ;
   BAR_5_E_ULASTI : BOOL ;
   JEN1_HAZIR : BOOL ;
   ANA_HAT_TRASFER_HAZIR : BOOL ;
   JEN_STATUS_REAL : INT ;
   STOP_SET_RESET : BOOL ;
   CALISMA_SURESI_TIME : TIME ;
   CALISMA_SURESI_DINT : DINT ;
   KRITIK_DEGERLERE_ULASTI : BOOL ;	//180 derece baca-6 bari gecti- 165 ic sicaklik
   CALISMA_SURESI_EKRAN : DINT ;
   SET2_DEGERINE_ULASMADI : BOOL ;
  END_STRUCT ;	
BEGIN
END_DATA_BLOCK

DATA_BLOCK DB 20
VERSION : 0.1
  STRUCT
   BASINC_SET_POINT : REAL ;
   STATUS : INT ;
   SICAKLIK_SET_POINT_1 : REAL ;
   SICAKLIK_SET_POINT_2 : REAL ;
   JEN2_SISTEM_BASLADI : BOOL ;
   EKRAN_START : BOOL ;
   EKRAN_STOP : BOOL ;
   OUT_BURLOR_MOT_START : BOOL ;
   SICAKLIK_SET1_OK : BOOL ;
   SICAKLIK_SET2_OK : BOOL ;
   OUT_PID_START : BOOL ;
   FAZ_GECISI_STATUS : INT ;
   FAZ_2_SET_RESET : BOOL ;
   BAR_5_E_ULASTI : BOOL ;
   JEN2_HAZIR : BOOL ;
   ANA_HAT_TRASNFER : BOOL ;
   JEN_STATUS_REAL : INT ;
   STOP_SET_RESET : BOOL ;
   CALISMA_SURESI_TIME : TIME ;
   CALISMA_SURESI_DINT : DINT ;
   KRITIK_DEGERE_ULASTI : BOOL ;	//Baca 180 derecede-6 bari gecti-165 ic sicaklik
   CALISMA_SURESI_EKRAN : DINT ;
  END_STRUCT ;	
BEGIN
END_DATA_BLOCK

DATA_BLOCK DB 21
VERSION : 0.1
  STRUCT
   TCONT_C_LMN : REAL ;
   TCONT_C_LMN_PER : INT ;
  END_STRUCT ;	
BEGIN
END_DATA_BLOCK

DATA_BLOCK DB 22
VERSION : 0.1
  STRUCT
   TCONT_C_LMN : REAL ;
   TCONT_C_LMN_PER : INT ;
  END_STRUCT ;	
BEGIN
END_DATA_BLOCK

DATA_BLOCK DB 23
VERSION : 0.1
  STRUCT
   TCONT_LMN_PER : INT ;
   TCONT_LMN : REAL ;
  END_STRUCT ;	
BEGIN
END_DATA_BLOCK

DATA_BLOCK DB 24
VERSION : 0.1
  STRUCT
   TCONT_LMN_PER : INT ;
   TCONT_LMN : REAL ;
  END_STRUCT ;	
BEGIN
END_DATA_BLOCK

DATA_BLOCK DB 50
AUTHOR : SIMATIC
FAMILY : ICONT
VERSION : 0.0
FB 41
BEGIN
END_DATA_BLOCK

DATA_BLOCK DB 51
VERSION : 0.0
FB 50
BEGIN
END_DATA_BLOCK

DATA_BLOCK DB 52
VERSION : 0.0
FB 49
BEGIN
END_DATA_BLOCK

DATA_BLOCK DB 69
AUTHOR : SIMATIC
FAMILY : CONTROL
VERSION : 0.0
FB 58
BEGIN
END_DATA_BLOCK

DATA_BLOCK DB 70
AUTHOR : SIMATIC
FAMILY : CONTROL
VERSION : 0.0
FB 58
BEGIN
END_DATA_BLOCK

DATA_BLOCK DB 94
VERSION : 0.0
FB 94
BEGIN
END_DATA_BLOCK

DATA_BLOCK DB 95
VERSION : 0.0
FB 95
BEGIN
END_DATA_BLOCK

DATA_BLOCK DB 98
VERSION : 0.0
FB 98
BEGIN
END_DATA_BLOCK

DATA_BLOCK DB 99
VERSION : 0.0
FB 99
BEGIN
END_DATA_BLOCK

DATA_BLOCK DB 100
VERSION : 0.1
  STRUCT
   JEN1_Min_Basinc : REAL  := 5.000000e+000;	//Jenerator 1 min otomatik sekans basinci
   JEN1_Max_Basinc : REAL  := 5.500000e+000;	//Jenerator 1 max otomatik sekans basinci
   JEN2_Min_Basinc : REAL  := 5.000000e+000;	//Jenerator 2 min otomatik sekans basinci
   JEN2_Max_Basinc : REAL  := 5.500000e+000;	//Jenerator 2 max otomatik sekans basinci
   OTOKLAV_First_Oran : REAL  := 2.000000e+001;	//Otoklav oransal vana otomatik sekans ilk acilis orani
   OTOKLAV_Kademeli_Artis : REAL ;	//Otoklav oransal vana kademeli artis katsayisi
  END_STRUCT ;	
BEGIN
   JEN1_Min_Basinc := 5.000000e+00;
   JEN1_Max_Basinc := 5.500000e+00;
   JEN2_Min_Basinc := 5.000000e+00;
   JEN2_Max_Basinc := 5.500000e+00;
END_DATA_BLOCK

DATA_BLOCK DB 120
VERSION : 0.0
FB 20
BEGIN
END_DATA_BLOCK

DATA_BLOCK DB 130
AUTHOR : SIMATIC
FAMILY : CONTROL
VERSION : 0.0
FB 58
BEGIN
END_DATA_BLOCK

DATA_BLOCK DB 131
VERSION : 0.0
FB 47
BEGIN
END_DATA_BLOCK

DATA_BLOCK DB 132
VERSION : 0.0
FB 48
BEGIN
END_DATA_BLOCK

DATA_BLOCK DB 230
VERSION : 0.0
FB 20
BEGIN
END_DATA_BLOCK

DATA_BLOCK DB 231
AUTHOR : SIMATIC
FAMILY : CONTROL
VERSION : 0.0
FB 58
BEGIN
END_DATA_BLOCK

DATA_BLOCK DB 232
VERSION : 0.0
FB 5
BEGIN
END_DATA_BLOCK

ORGANIZATION_BLOCK OB 1
TITLE = "Main Program Sweep (Cycle)"
VERSION : 0.1
VAR_TEMP
  OB1_EV_CLASS : BYTE ;	//Bits 0-3 = 1 (Coming event), Bits 4-7 = 1 (Event class 1)
  OB1_SCAN_1 : BYTE ;	//1 (Cold restart scan 1 of OB 1), 3 (Scan 2-n of OB 1)
  OB1_PRIORITY : BYTE ;	//Priority of OB Execution
  OB1_OB_NUMBR : BYTE ;	//1 (Organization block 1, OB1)
  OB1_RESERVED_1 : BYTE ;	//Reserved for system
  OB1_RESERVED_2 : BYTE ;	//Reserved for system
  OB1_PREV_CYCLE : INT ;	//Cycle time of previous OB1 scan (milliseconds)
  OB1_MIN_CYCLE : INT ;	//Minimum cycle time of OB1 (milliseconds)
  OB1_MAX_CYCLE : INT ;	//Maximum cycle time of OB1 (milliseconds)
  OB1_DATE_TIME : DATE_AND_TIME ;	//Date and time OB1 started
END_VAR
BEGIN
NETWORK
TITLE = ALWAYS OFF
      UC    FB 1;
NETWORK
TITLE = HAVA VE HAT BASINCI
      CALL  FC 105 (
           $1                       := P#P 292.0,
           $2                       := L#1092616192,
           $3                       := L#0,
           $4                       := P#M 100.0,
           $5                       := DB1.DBW 36,
           $6                       := DB1.DBD 38);
      CALL  FC 105 (
           $1                       := P#P 294.0,
           $2                       := L#1092616192,
           $3                       := L#0,
           $4                       := P#M 100.0,
           $5                       := DB1.DBW 42,
           $6                       := DB1.DBD 44);
NETWORK
TITLE = ACIKLAMALAR
//FB98 - JEN 1 KONTROL BLOGU
//FB99 - JEN 2 KONTROL BLOGU
//FB49 - JEN 1 PID KONTROL - PID BLOKLARI
//FB50 - JEN 2 PID KONTROL - PID BLOKLARI
//FB94 - KAZAN 1 KONTROL BLOGU - KAZAN 1 ILE ILGILI KONTROLLER
//FB95 - KAZAN 2 KONTROL BLOGU - KAZAN 2 ILE ILGILI KONTROLLER
//FB47 - KAZAN 1 PID KONTROL
//FB48 - KAZAN 2 PID KONTROL
//FB3 - SURELER - KAZAN1,KAZAN2, JEN1, JEN2 ILE ILGILI TUM SURELER BURADA TUTULUR
//FB2 - SAFETY
//      1)JEN1, JEN2 KRITIK SU SEVIYE MIKTARLARI
//      2)HAVA BASINCI KONTROLU
//      3)JENERATOR IS BITIMINDE BORUDA KALAN BUHARIN TAHLIYESI
//FB1 - MAINBLOCK  
//      1)ÇALISACAK TUM BLOKLAR BURADA CAGRILIR
//      2)AYRICA HAVA VE HAT BASINCI DONUSUMLARI BURADADIR
//FB5 - TEST BLOGU - PROSESIN DEVREYE ALINAMADAN ONCEKI TEST ISLEMLERININ GERCEKLESTIGI
//      BLOKTUR.
END_ORGANIZATION_BLOCK

ORGANIZATION_BLOCK OB 35
TITLE = "Cyclic Interrupt"
VERSION : 0.1
VAR_TEMP
  OB35_EV_CLASS : BYTE ;	//Bits 0-3 = 1 (Coming event), Bits 4-7 = 1 (Event class 1)
  OB35_STRT_INF : BYTE ;	//16#36 (OB 35 has started)
  OB35_PRIORITY : BYTE ;	//Priority of OB Execution
  OB35_OB_NUMBR : BYTE ;	//35 (Organization block 35, OB35)
  OB35_RESERVED_1 : BYTE ;	//Reserved for system
  OB35_RESERVED_2 : BYTE ;	//Reserved for system
  OB35_PHASE_OFFSET : WORD ;	//Phase offset (msec)
  OB35_RESERVED_3 : INT ;	//Reserved for system
  OB35_EXC_FREQ : INT ;	//Frequency of execution (msec)
  OB35_DATE_TIME : DATE_AND_TIME ;	//Date and time OB35 started
END_VAR
BEGIN
NETWORK
TITLE =
      CALL  FB 49 , DB 52;
      CALL  FB 50 , DB 51;
NETWORK
TITLE =
      CALL  FB 47 , DB 131;
      CALL  FB 48 , DB 132;
END_ORGANIZATION_BLOCK

ORGANIZATION_BLOCK OB 80
TITLE = "Cycle Time Fault"
VERSION : 0.1
VAR_TEMP
  OB80_EV_CLASS : BYTE ;	//16#35, Event class 3, Entering event state, Internal fault event
  OB80_FLT_ID : BYTE ;	//16#XX, Fault identifcation code
  OB80_PRIORITY : BYTE ;	//Priority of OB Execution
  OB80_OB_NUMBR : BYTE ;	//80 (Organization block 80, OB80)
  OB80_RESERVED_1 : BYTE ;	//Reserved for system
  OB80_RESERVED_2 : BYTE ;	//Reserved for system
  OB80_ERROR_INFO : WORD ;	//Error information on event
  OB80_ERR_EV_CLASS : BYTE ;	//Class of event causing error
  OB80_ERR_EV_NUM : BYTE ;	//Number of event causing error
  OB80_OB_PRIORITY : BYTE ;	//Priority of OB causing error
  OB80_OB_NUM : BYTE ;	//Number of OB causing error
  OB80_DATE_TIME : DATE_AND_TIME ;	//Date and time OB80 started
END_VAR
BEGIN
// (block stored without names or comments; labels and parameter names are numbered)
END_ORGANIZATION_BLOCK

ORGANIZATION_BLOCK OB 81
TITLE = "Power Supply Fault"
VERSION : 0.1
VAR_TEMP
  OB81_EV_CLASS : BYTE ;	//16#39, Event class 3, Entering event state, Internal fault event
  OB81_FLT_ID : BYTE ;	//16#XX, Fault identifcation code
  OB81_PRIORITY : BYTE ;	//Priority of OB Execution
  OB81_OB_NUMBR : BYTE ;	//81 (Organization block 81, OB81)
  OB81_RESERVED_1 : BYTE ;	//Reserved for system
  OB81_RESERVED_2 : BYTE ;	//Reserved for system
  OB81_RACK_CPU : WORD ;	//see online help (F1)
  OB81_RESERVED_3 : BYTE ;	//Reserved for system
  OB81_RESERVED_4 : BYTE ;	//Reserved for system
  OB81_RESERVED_5 : BYTE ;	//Reserved for system
  OB81_RESERVED_6 : BYTE ;	//Reserved for system
  OB81_DATE_TIME : DATE_AND_TIME ;	//Date and time OB81 started
END_VAR
BEGIN
// (block stored without names or comments; labels and parameter names are numbered)
END_ORGANIZATION_BLOCK

ORGANIZATION_BLOCK OB 82
TITLE = "I/O Point Fault"
VERSION : 0.1
VAR_TEMP
  OB82_EV_CLASS : BYTE ;	//16#39, Event class 3, Entering event state, Internal fault event
  OB82_FLT_ID : BYTE ;	//16#XX, Fault identifcation code
  OB82_PRIORITY : BYTE ;	//Priority of OB Execution
  OB82_OB_NUMBR : BYTE ;	//82 (Organization block 82, OB82)
  OB82_RESERVED_1 : BYTE ;	//Reserved for system
  OB82_IO_FLAG : BYTE ;	//Input (01010100), Output (01010101)
  OB82_MDL_ADDR : WORD ;	//Base address of module with fault
  OB82_MDL_DEFECT : BOOL ;	//Module defective
  OB82_INT_FAULT : BOOL ;	//Internal fault
  OB82_EXT_FAULT : BOOL ;	//External fault
  OB82_PNT_INFO : BOOL ;	//Point information
  OB82_EXT_VOLTAGE : BOOL ;	//External voltage low
  OB82_FLD_CONNCTR : BOOL ;	//Field wiring connector missing
  OB82_NO_CONFIG : BOOL ;	//Module has no configuration data
  OB82_CONFIG_ERR : BOOL ;	//Module has configuration error
  OB82_MDL_TYPE : BYTE ;	//Type of module
  OB82_SUB_MDL_ERR : BOOL ;	//Sub-Module is missing or has error
  OB82_COMM_FAULT : BOOL ;	//Communication fault
  OB82_MDL_STOP : BOOL ;	//Module is stopped
  OB82_WTCH_DOG_FLT : BOOL ;	//Watch dog timer stopped module
  OB82_INT_PS_FLT : BOOL ;	//Internal power supply fault
  OB82_PRIM_BATT_FLT : BOOL ;	//Primary battery is in fault
  OB82_BCKUP_BATT_FLT : BOOL ;	//Backup battery is in fault
  OB82_RESERVED_2 : BOOL ;	//Reserved for system
  OB82_RACK_FLT : BOOL ;	//Rack fault, only for bus interface module
  OB82_PROC_FLT : BOOL ;	//Processor fault
  OB82_EPROM_FLT : BOOL ;	//EPROM fault
  OB82_RAM_FLT : BOOL ;	//RAM fault
  OB82_ADU_FLT : BOOL ;	//ADU fault
  OB82_FUSE_FLT : BOOL ;	//Fuse fault
  OB82_HW_INTR_FLT : BOOL ;	//Hardware interupt input in fault
  OB82_RESERVED_3 : BOOL ;	//Reserved for system
  OB82_DATE_TIME : DATE_AND_TIME ;	//Date and time OB82 started
END_VAR
BEGIN
// (block stored without names or comments; labels and parameter names are numbered)
END_ORGANIZATION_BLOCK

ORGANIZATION_BLOCK OB 83
TITLE = "I/O Point Fault"
VERSION : 0.1
VAR_TEMP
  OB83_EV_CLASS : BYTE ;	//16#38/39, Event class 3, module inserted/removed (8/9)
  OB83_FLT_ID : BYTE ;	//16#XX, Fault identifcation code
  OB83_PRIORITY : BYTE ;	//Priority of OB Execution
  OB83_OB_NUMBR : BYTE ;	//83 (Organization block 83, OB83)
  OB83_RESERVED_1 : BYTE ;	//Reserved for system
  OB83_MDL_ID : BYTE ;	//Input module (01010100), Output module (01010101)
  OB83_MDL_ADDR : WORD ;	//Base address of module with point fault
  OB83_RACK_NUM : INT ;	//Number of rack that has module with point fault
  OB83_MDL_TYPE : WORD ;	//Module type with point fault
  OB83_DATE_TIME : DATE_AND_TIME ;	//Date and time OB83 started
END_VAR
BEGIN
// (block stored without names or comments; labels and parameter names are numbered)
END_ORGANIZATION_BLOCK

ORGANIZATION_BLOCK OB 84
TITLE = "CPU Fault"
VERSION : 0.1
VAR_TEMP
  OB84_EV_CLASS : BYTE ;	//16#38/39, Event class 3, module inserted/removed (8/9)
  OB84_FLT_ID : BYTE ;	//16#81, Fault identifcation code
  OB84_PRIORITY : BYTE ;	//Priority of OB Execution
  OB84_OB_NUMBR : BYTE ;	//84 (Organization block 84, OB84)
  OB84_RESERVED_1 : BYTE ;	//Reserved for system
  OB84_RESERVED_2 : BYTE ;	//Reserved for system
  OB84_RESERVED_3 : WORD ;	//Reserved for system
  OB84_RESERVED_4 : DWORD ;	//Reserved for system
  OB84_DATE_TIME : DATE_AND_TIME ;	//Date and time OB84 started
END_VAR
BEGIN
// (block stored without names or comments; labels and parameter names are numbered)
END_ORGANIZATION_BLOCK

ORGANIZATION_BLOCK OB 85
TITLE = "Organization Block (OB) Not Loaded Fault"
VERSION : 0.1
VAR_TEMP
  OB85_EV_CLASS : BYTE ;	//16#35 Event class 3
  OB85_FLT_ID : BYTE ;	//16#XX, Fault identification code
  OB85_PRIORITY : BYTE ;	//Priority of OB Execution
  OB85_OB_NUMBR : BYTE ;	//85 (Organization block 85, OB85)
  OB85_RESERVED_1 : BYTE ;	//Reserved for system
  OB85_RESERVED_2 : BYTE ;	//Reserved for system
  OB85_RESERVED_3 : INT ;	//Reserved for system
  OB85_ERR_EV_CLASS : BYTE ;	//Class of event causing error
  OB85_ERR_EV_NUM : BYTE ;	//Number of event causing error
  OB85_OB_PRIOR : BYTE ;	//Priority of OB causing error
  OB85_OB_NUM : BYTE ;	//Number of OB causing error
  OB85_DATE_TIME : DATE_AND_TIME ;	//Date and time OB85 started
END_VAR
BEGIN
// (block stored without names or comments; labels and parameter names are numbered)
END_ORGANIZATION_BLOCK

ORGANIZATION_BLOCK OB 86
TITLE = "Loss Of Rack Fault"
VERSION : 0.1
VAR_TEMP
  OB86_EV_CLASS : BYTE ;	//16#38/39 Event class 3
  OB86_FLT_ID : BYTE ;	//16#C1/C4/C5, Fault identifcation code
  OB86_PRIORITY : BYTE ;	//Priority of OB Execution
  OB86_OB_NUMBR : BYTE ;	//86 (Organization block 86, OB86)
  OB86_RESERVED_1 : BYTE ;	//Reserved for system
  OB86_RESERVED_2 : BYTE ;	//Reserved for system
  OB86_MDL_ADDR : WORD ;	//Base address of IM module in rack with fault
  OB86_RACKS_FLTD : ARRAY  [0 .. 31 ] OF BOOL ;	//Racks in fault
  OB86_DATE_TIME : DATE_AND_TIME ;	//Date and time OB86 started
END_VAR
BEGIN
// (block stored without names or comments; labels and parameter names are numbered)
END_ORGANIZATION_BLOCK

ORGANIZATION_BLOCK OB 87
TITLE = "Communication Fault"
VERSION : 0.1
VAR_TEMP
  OB87_EV_CLASS : BYTE ;	//16#39 Event class 3
  OB87_FLT_ID : BYTE ;	//16#XX, Fault identifcation code
  OB87_PRIORITY : BYTE ;	//Priority of OB Execution
  OB87_OB_NUMBR : BYTE ;	//87 (Organization block 87, OB87)
  OB87_RESERVED_1 : BYTE ;	//Reserved for system
  OB87_RESERVED_2 : BYTE ;	//Reserved for system
  OB87_RESERVED_3 : WORD ;	//Reserved for system
  OB87_RESERVED_4 : DWORD ;	//Reserved for system
  OB87_DATE_TIME : DATE_AND_TIME ;	//Date and time OB87 started
END_VAR
BEGIN
// (block stored without names or comments; labels and parameter names are numbered)
END_ORGANIZATION_BLOCK

ORGANIZATION_BLOCK OB 100
TITLE = "Complete Restart"
VERSION : 0.1
VAR_TEMP
  OB100_EV_CLASS : BYTE ;	//16#13, Event class 1, Entering event state, Event logged in diagnostic buffer
  OB100_STRTUP : BYTE ;	//16#81/82/83/84 Method of startup
  OB100_PRIORITY : BYTE ;	//Priority of OB Execution
  OB100_OB_NUMBR : BYTE ;	//100 (Organization block 100, OB100)
  OB100_RESERVED_1 : BYTE ;	//Reserved for system
  OB100_RESERVED_2 : BYTE ;	//Reserved for system
  OB100_STOP : WORD ;	//Event that caused CPU to stop (16#4xxx)
  OB100_STRT_INFO : DWORD ;	//Information on how system started
  OB100_DATE_TIME : DATE_AND_TIME ;	//Date and time OB100 started
END_VAR
BEGIN
NETWORK
TITLE = Kazan islemlerini sifirlama islemleri
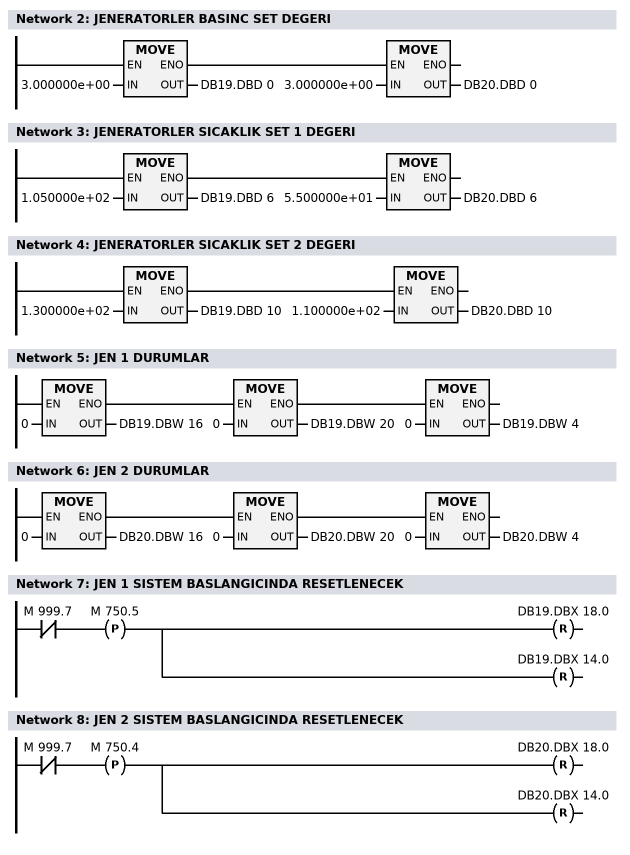
NETWORK
TITLE = JENERATORLER BASINC SET DEGERI
      A(;
      L     3.000000e+00;
      T     DB19.DBD 0;
      SET;
      SAVE;
      CLR;
      A     BR;
      );
      JNB   _001;
      L     3.000000e+00;
      T     DB20.DBD 0;
_001: NOP   0;
NETWORK
TITLE = JENERATORLER SICAKLIK SET 1 DEGERI
      A(;
      L     1.050000e+02;
      T     DB19.DBD 6;
      SET;
      SAVE;
      CLR;
      A     BR;
      );
      JNB   _002;
      L     5.500000e+01;
      T     DB20.DBD 6;
_002: NOP   0;
NETWORK
TITLE = JENERATORLER SICAKLIK SET 2 DEGERI
      A(;
      L     1.300000e+02;
      T     DB19.DBD 10;
      SET;
      SAVE;
      CLR;
      A     BR;
      );
      JNB   _003;
      L     1.100000e+02;
      T     DB20.DBD 10;
_003: NOP   0;
NETWORK
TITLE = JEN 1 DURUMLAR
      A(;
      A(;
      L     0;
      T     DB19.DBW 16;
      SET;
      SAVE;
      CLR;
      A     BR;
      );
      JNB   _004;
      L     0;
      T     DB19.DBW 20;
      SET;
      SAVE;
      CLR;
_004: A     BR;
      );
      JNB   _005;
      L     0;
      T     DB19.DBW 4;
_005: NOP   0;
NETWORK
TITLE = JEN 2 DURUMLAR
      A(;
      A(;
      L     0;
      T     DB20.DBW 16;
      SET;
      SAVE;
      CLR;
      A     BR;
      );
      JNB   _006;
      L     0;
      T     DB20.DBW 20;
      SET;
      SAVE;
      CLR;
_006: A     BR;
      );
      JNB   _007;
      L     0;
      T     DB20.DBW 4;
_007: NOP   0;
NETWORK
TITLE = JEN 1 SISTEM BASLANGICINDA RESETLENECEK
      AN    M 999.7;
      FP    M 750.5;
      R     DB19.DBX 18.0;
      R     DB19.DBX 14.0;
NETWORK
TITLE = JEN 2 SISTEM BASLANGICINDA RESETLENECEK
      AN    M 999.7;
      FP    M 750.4;
      R     DB20.DBX 18.0;
      R     DB20.DBX 14.0;
END_ORGANIZATION_BLOCK

ORGANIZATION_BLOCK OB 101
TITLE = "Restart"
VERSION : 0.1
VAR_TEMP
  OB101_EV_CLASS : BYTE ;	//16#13, Event class 1, Entering event state, Event logged in diagnostic buffer
  OB101_STRTUP : BYTE ;	//16#81/82/83/84 Method of startup
  OB101_PRIORITY : BYTE ;	//Priority of OB Execution
  OB101_OB_NUMBR : BYTE ;	//101 (Organization block 101, OB101)
  OB101_RESERVED_1 : BYTE ;	//Reserved for system
  OB101_RESERVED_2 : BYTE ;	//Reserved for system
  OB101_STOP : WORD ;	//Event that caused CPU to stop (16#4xxx)
  OB101_STRT_INFO : DWORD ;	//Information on how system started
  OB101_DATE_TIME : DATE_AND_TIME ;	//Date and time OB101 started
END_VAR
BEGIN
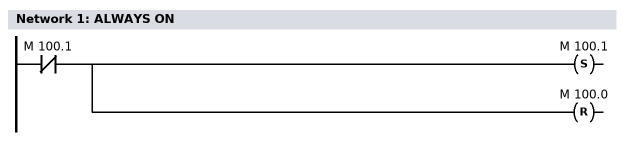
NETWORK
TITLE = ALWAYS ON
      AN    M 100.1;
      S     M 100.1;
      R     M 100.0;
END_ORGANIZATION_BLOCK

ORGANIZATION_BLOCK OB 102
TITLE = "Cold Restart"
VERSION : 0.1
VAR_TEMP
  OB102_EV_CLASS : BYTE ;	//16#13, Event class 1, Entering event state, Event logged in diagnostic buffer
  OB102_STRTUP : BYTE ;	//16#85...8B Method of startup
  OB102_PRIORITY : BYTE ;	//Priority of OB Execution
  OB102_OB_NUMBR : BYTE ;	//102 (Organization block 102, OB102)
  OB102_RESERVED_1 : BYTE ;	//Reserved for system
  OB102_RESERVED_2 : BYTE ;	//Reserved for system
  OB102_STOP : WORD ;	//Event that caused CPU to stop (16#4xxx)
  OB102_STRT_INFO : DWORD ;	//Information on how system started
  OB102_DATE_TIME : DATE_AND_TIME ;	//Date and time OB102 started
END_VAR
BEGIN
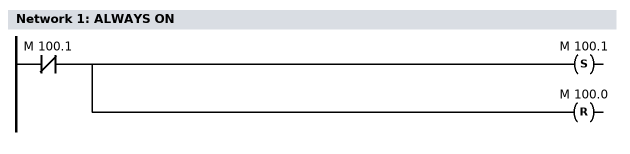
NETWORK
TITLE = ALWAYS ON
      AN    M 100.1;
      S     M 100.1;
      R     M 100.0;
END_ORGANIZATION_BLOCK

ORGANIZATION_BLOCK OB 121
TITLE = "Programming Error"
VERSION : 0.1
VAR_TEMP
  OB121_EV_CLASS : BYTE ;	//16#25, Event class 2, Entering event state, Internal fault event
  OB121_SW_FLT : BYTE ;	//16#XX Software programming fault
  OB121_PRIORITY : BYTE ;	//Priority of OB Execution
  OB121_OB_NUMBR : BYTE ;	//121 (Organization block 121, OB121)
  OB121_BLK_TYPE : BYTE ;	//16#88/8A/8B/8C/8E Type of block fault occured in
  OB121_RESERVED_1 : BYTE ;	//Reserved for system
  OB121_FLT_REG : WORD ;	//16#XX Specific register that caused fault
  OB121_BLK_NUM : WORD ;	//Number of block that programming fault occured in
  OB121_PRG_ADDR : WORD ;	//Address in block where programming fault occured
  OB121_DATE_TIME : DATE_AND_TIME ;	//Date and time OB121 started
END_VAR
BEGIN
// (block stored without names or comments; labels and parameter names are numbered)
END_ORGANIZATION_BLOCK

SYMBOL_TABLE
"AI-SENSOR-DATA"	DB 1	DB 1
"ORTAK_DATA"	DB 2	DB 2	// Ortak Veriler
"TIME_OTO_1_DB"	DB 5	SFB 4
"TIME_OTO_2_DB"	DB 6	SFB 4
"TIME_OTO_1_PROSES_DB"	DB 7	SFB 4
"TIME_OTO_2_PROSES_DB"	DB 8	SFB 4
"SURELER_DB"	DB 14	FB 3
"SAFETY_DB"	DB 15	FB 2
"KAZAN1_DATA"	DB 17	DB 17
"KAZAN2_DATA"	DB 18	DB 18	// KAZAN 2 BILGILERI
"JEN1_DATA"	DB 19	DB 19
"JEN2_DATA"	DB 20	DB 20
"JEN1_PID_DATA"	DB 21	DB 21
"JEN2_PID_DATA"	DB 22	DB 22
"KAZAN1_PID_DATA"	DB 23	DB 23	// KAZAN 1 PID BILGILERI
"KAZAN2_PID_DATA"	DB 24	DB 24	// KAZAN 2 PID BILGILERI
"JEN2_KONTROL_BLOGU_DB"	DB 51	FB 50
"JEN_1_PID_DB"	DB 69	FB 58
"JEN_2_PID_DB"	DB 70	FB 58
"OTOKLAV_1_DB"	DB 94	FB 94
"OTOKLAV_2_DB"	DB 95	FB 95
"FB98_DB"	DB 98	FB 98
"FB99_DB"	DB 99	FB 99
"HMI_DATA"	DB 100	DB 100	// Hmi arayuz verileri
"KAZAN_1_PID_DB"	DB 130	FB 58
"KAZAN_2_PID_DATA"	DB 231	FB 58
"MAINBLOCK"	FB 1	FB 1	// ANA PROGRAM BLOGU
"SAFETY"	FB 2	FB 2
"SURELER"	FB 3	FB 3
"TEST_BLOGU"	FB 5	FB 5
"KAZAN_ORTAK"	FB 20	FB 20
"CONT_C"	FB 41	FB 41	// Continuous Control
"KAZAN_1_PID_KONTROL"	FB 47	FB 47
"KAZAN_2_PID_KONTROL"	FB 48	FB 48
"JEN1_PID_KONTROL"	FB 49	FB 49
"JEN2_PID_KONTROL"	FB 50	FB 50	// BUAHR JENERATÖR 2 PID
"TCONT_CP"	FB 58	FB 58	// temperature PID controller with pulse generator and self-tuning
"KAZAN_1_KONTROL"	FB 94	FB 94
"KAZAN_2_KONTROL"	FB 95	FB 95
"JEN1_KONTROL_BLOGU"	FB 98	FB 98
"JEN2_KONTROL_BLOGU"	FB 99	FB 99
"TIME_UNSCALE"	FC 1	FC 1
"S5TI_TIM"	FC 33	FC 33	// S5 Time to IEC Time
"SCALE"	FC 105	FC 105	// Scaling Values
"UNSCALE"	FC 106	FC 106	// Unscaling Values
"PID BLOCK"	OB 35	OB 35	// PID BLOCK
"ZAMANHATASI"	OB 80	OB 80	// ZAMAN HATASI
"GERILIMHATASI"	OB 81	OB 81	// BESLEME GERILIMI HATASI
"HATAUYARISI"	OB 82	OB 82	// HATA UYARISI
"TAKMACIKARMAHATASI"	OB 83	OB 83	// TAKMA ÇIKARMA UYARISI
"CPUHARDWAREERROR"	OB 84	OB 84	// CPU HARDWARE ERROR
"PROGRAMHATASI"	OB 85	OB 85	// PROGRAM YURUTME HATASI
"RACKHATASI"	OB 86	OB 86	// RACK HATASI
"HABERLESMEHATASI"	OB 87	OB 87	// HABERLESME HATASI,
"COMPLETE RESTART"	OB 100	OB 100	// Complete Restart
"RESTART"	OB 101	OB 101	// Restart
"COLD RESTART"	OB 102	OB 102	// Cold Restart
"PROGRAMMINGERROR"	OB 121	OB 121	// PROGRAMLAMA HATASI
"TON"	SFB 4	SFB 4	// Generate an On Delay
"TEST BLOGU VAT"	VAT 1	
"JEN2_MONITOR"	VAT 2	
"KAZAN-1-MONITOR"	VAT 3	
"KAZAN-2-MONITOR"	VAT 4	
"JEN1_MONITOR"	VAT 5	
"deneme"	VAT 6	
END_SYMBOL_TABLE
